{attribute 'qualified_only'}
{attribute 'strict'}
TYPE E_MC_STEP :
(
	Restart,
	Power,
	MoveAbs
);
END_TYPE

(* stored: Version 1.1.0.1, ProductVersion 3.1.4024.13
   DUT E_MC_STEP: Id {cef47bb7-116c-46bb-9cc4-88deadd8de25} *)
